SUBAPPLICATION Uebung_034b (* LONG_PRESS_HOLD-Eingang auf PWM Ausgang mit Terminal-Ausgabe *)
  (* Standard: 61499-2; Description: Copyright (c) 2023 Meisterschulen am Ostbahnhof This program and the accompanying materials are made available under the terms of the Eclipse Public License 2.0 which is available at https://www.eclipse.org/legal/epl-2.0/ SPDX-License-Identifier: EPL-2.0 *)
  (* Version 1.1, 2026-04-21, Franz Höpfinger, Meisterschulen am Ostbahnhof, Added terminal output for counter value *)
  (* Version 1.0, 2023-10-23, Franz Höpfinger, Meisterschulen am Ostbahnhof, initial API and implementation and/or initial documentation *)
  PACKAGE Uebungen;
  IMPORT Uebungen::const::UT::DefaultPool::OutputNumber_N1;
  IMPORT logiBUS::io::DI::logiBUS_DI::Input_I1;
  IMPORT logiBUS::io::DI::logiBUS_DI::Input_I2;
  IMPORT logiBUS::io::DI::logiBUS_DI::Input_I3;
  IMPORT logiBUS::io::DI::logiBUS_DI::Input_I4;
  IMPORT logiBUS::io::DI::logiBUS_DI_Events::BUTTON_LONG_PRESS_HOLD;
  IMPORT logiBUS::io::DI::logiBUS_DI_Events::BUTTON_SINGLE_CLICK;
  IMPORT logiBUS::io::DQ::logiBUS_DO::Output_Q1;
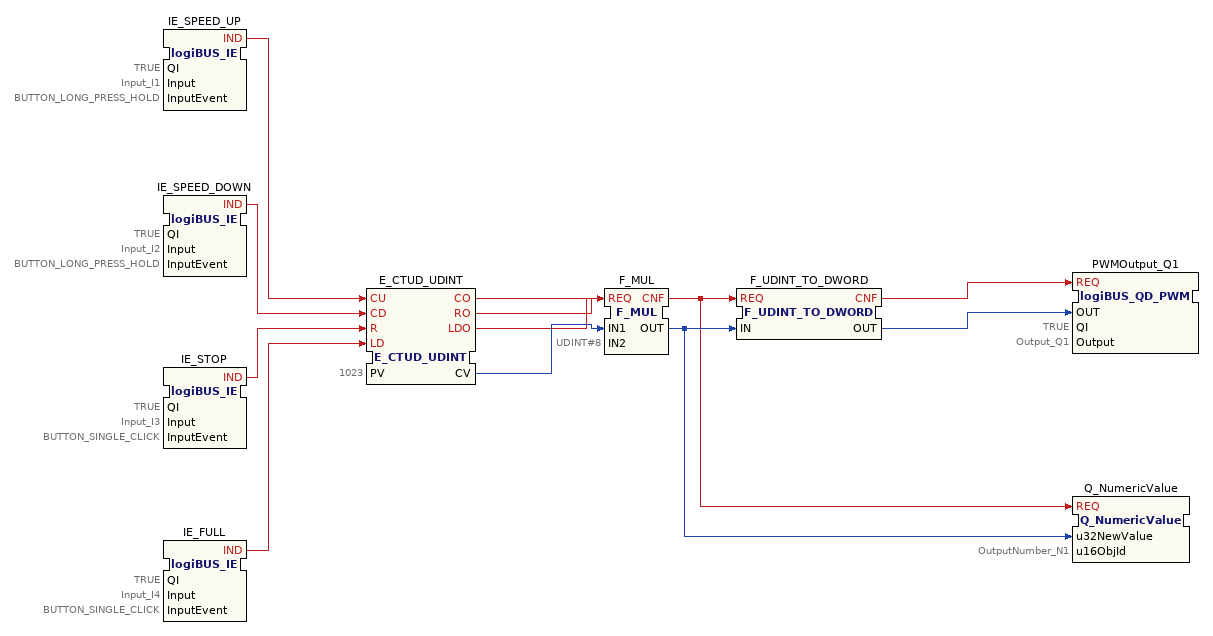
  FBS
    PWMOutput_Q1 : logiBUS::io::DQ::logiBUS_QD_PWM(QI := TRUE, Output := Output_Q1);
    IE_SPEED_UP : logiBUS::io::DI::logiBUS_IE(QI := TRUE, Input := Input_I1, InputEvent := BUTTON_LONG_PRESS_HOLD);
    IE_SPEED_DOWN : logiBUS::io::DI::logiBUS_IE(QI := TRUE, Input := Input_I2, InputEvent := BUTTON_LONG_PRESS_HOLD);
    E_CTUD_UDINT : iec61499::events::E_CTUD_UDINT(PV := 1023);
    F_UDINT_TO_DWORD : iec61131::conversion::F_UDINT_TO_DWORD;
    IE_STOP : logiBUS::io::DI::logiBUS_IE(QI := TRUE, Input := Input_I3, InputEvent := BUTTON_SINGLE_CLICK);
    IE_FULL : logiBUS::io::DI::logiBUS_IE(QI := TRUE, Input := Input_I4, InputEvent := BUTTON_SINGLE_CLICK);
    F_MUL : iec61131::arithmetic::F_MUL(IN2 := UDINT#8);
    Q_NumericValue : isobus::UT::Q::Q_NumericValue(u16ObjId := OutputNumber_N1);
  END_FBS
  EVENT_CONNECTIONS
    E_CTUD_UDINT.CO TO F_MUL.REQ;
    E_CTUD_UDINT.RO TO F_MUL.REQ;
    IE_SPEED_UP.IND TO E_CTUD_UDINT.CU;
    IE_SPEED_DOWN.IND TO E_CTUD_UDINT.CD;
    IE_STOP.IND TO E_CTUD_UDINT.R;
    IE_FULL.IND TO E_CTUD_UDINT.LD;
    E_CTUD_UDINT.LDO TO F_MUL.REQ;
    F_UDINT_TO_DWORD.CNF TO PWMOutput_Q1.REQ;
    F_MUL.CNF TO F_UDINT_TO_DWORD.REQ;
    F_MUL.CNF TO Q_NumericValue.REQ;
  END_CONNECTIONS
  DATA_CONNECTIONS
    E_CTUD_UDINT.CV TO F_MUL.IN1;
    F_UDINT_TO_DWORD.OUT TO PWMOutput_Q1.OUT;
    F_MUL.OUT TO F_UDINT_TO_DWORD.IN;
    F_MUL.OUT TO Q_NumericValue.u32NewValue;
  END_CONNECTIONS
END_SUBAPPLICATION
